FUNCTION_BLOCK FB_Restore
VAR_INPUT
	iMotorPrev 		: 	INT;
	eStep		:	E_Step;
	eSubStep	:	E_Step;
END_VAR
VAR_IN_OUT
	stIn		:	ST_CSL_In;
	stParams	: 	ST_CSL_Params;
	stOut		:	ST_CSL_Out;
END_VAR
VAR_OUTPUT
	bFbEnd		:	BOOL;
END_VAR
VAR
	iMotor		:	INT;

	bPieceOut 	:	BOOL;	

	fbRtMotorImpulse : R_TRIG;
END_VAR

IF eStep = E_Step.MainSensor THEN
	IF NOT stIn.bPieceSensorOutput AND NOT bPieceOut THEN
		stOut.bMotor := TRUE;
		bPieceOut := TRUE;
	END_IF
	IF bPieceOut THEN
		fbRtMotorImpulse(CLK:=	stIn.bMotorImpulse );
		
		IF fbRtMotorImpulse.Q	THEN
			iMotor := iMotor + 1;
		END_IF
			
		IF iMotor = stParams.StepNoSlot THEN
			stOut.bMotor := FALSE;
			bPieceOut	:=	FALSE;
			bFbEnd := TRUE;
		END_IF
		
	END_IF
	
ELSIF eStep = E_Step.MainPiston THEN
	stOut.bMotor := TRUE;
	
	fbRtMotorImpulse(CLK:=	stIn.bMotorImpulse );
		
	IF fbRtMotorImpulse.Q	THEN
		iMotor := iMotor + 1;
	END_IF
			
	IF iMotor = (stParams.StepNoSlot - iMotorPrev + 1) THEN
		stOut.bMotor := FALSE;
		bFbEnd := TRUE;
	END_IF

ELSE
	IF stIn.bPieceSensorInput AND stIn.bPieceSensorOutput AND stIn.bSlot1 AND stIn.bSlot2 AND stIn.bSlot3 THEN 
		bFbEnd := TRUE;
	END_IF
END_IF

END_FUNCTION_BLOCK

(* stored: Version 1.1.0.1, ProductVersion 3.1.4024.12
   POU FB_Restore: Id {fd15dcd7-03bd-4602-ba28-f37f0729ceb4}, SpecialFunc None *)
